// TIA Portal V14 export
ORGANIZATION_BLOCK "Main"   // OB1, SCL
// stored: AutoNumber true
BEGIN
END_ORGANIZATION_BLOCK
